// TIA Portal V19 export
DATA_BLOCK "DEBUG_MES_Receive_Msg_Topic2XX"   // DB204
// stored: MemoryReserve 100
   VAR
      DEBUG { ExternalAccessible := 'False'; ExternalVisible := 'False'; ExternalWritable := 'False'} : Struct
         Enable : Bool;
         AckChangeStep : Bool;
         ActualStep : Int;
      END_STRUCT;
      ACK_MSG_enable : Bool;
      MSG_200 : Struct
         ABILITA_FC : Bool;
         EXE_MSG : Bool;
         MSG : "MES_Msg";
      END_STRUCT;
      MSG_210 : Struct
         ABILITA_FC : Bool;
         EXE_MSG : Bool;
         MSG : "MES_Msg";
      END_STRUCT;
      MSG_212 : Struct
         ABILITA_FC : Bool;
         EXE_MSG : Bool;
         MSG : "MES_Msg";
      END_STRUCT;
   END_VAR
BEGIN
END_DATA_BLOCK
